PROGRAM P_Demo_FB_DMXGetDeviceLabel
VAR
    fbGetDeviceLabel  : FB_DMXGetDeviceLabel;         // 读设备标签
    stDmxCmdBuffer    : ST_DMXCommandBuffer;          // 与通讯 FB 共用
    wTargetManufId    : WORD := 16#4241;              // 目标灯具厂商 ID
    dwTargetDeviceId  : DWORD := 16#12131415;         // 目标灯具设备 ID
    byTargetPort      : BYTE := 0;                    // 根设备通道 0
    bDoRead           : BOOL := FALSE;                // 在线给一次上升沿触发
    bBusy             : BOOL;
    bError            : BOOL;
    udiErrId          : UDINT;
    sLabel            : STRING;                       // 设备标签文本
END_VAR

// ============================================================
// Tc2_DMX.FB_DMXGetDeviceLabel 演示程序
// ============================================================
// 场景：HMI 设备列表显示：把每盏灯在设备里存的自定义标签读出显示，让运维一眼辨识具体哪台。
// 价值：把人为可读的设备名读进 HMI，提升运维可读性，命名信息随设备走（换 PLC 也不丢）。
// 验证：先用 FB_DMXSetDeviceLabel 写一个标签，再给 bDoRead 一次上升沿 -> bBusy 短暂 TRUE -> 回 FALSE 后 sLabel 应等于所写文本。
// 验证步骤：
//   1. 右键 PLC 项目下 POUs 文件夹 → Add → Existing Item → 选本 .TcPOU 文件
//   2. 引用 Tc2_DMX；同项目里放一个 FB_EL6851CommunicationEx 实例并共用 stDmxCmdBuffer（非 CycleMode）
//   3. 编译 → 登录 → 运行；按上方『验证』行在线给上升沿观察
// ============================================================

fbGetDeviceLabel(
    bStart                     := bDoRead,
    wDestinationManufacturerId := wTargetManufId,
    dwDestinationDeviceId      := dwTargetDeviceId,
    byPortId                   := byTargetPort,
    dwOptions                  := 0,
    stCommandBuffer            := stDmxCmdBuffer,
    bBusy                      => bBusy,
    bError                     => bError,
    udiErrorId                 => udiErrId,
    sDeviceLabel               => sLabel
);

END_PROGRAM

(* stored: Version 1.1.0.1, ProductVersion 3.1.4024.5
   POU P_Demo_FB_DMXGetDeviceLabel: Id {8e76b4c8-7f63-58e9-a7f2-386a57af3d1d}, SpecialFunc None *)
